FUNCTION LogMessage
VAR_INPUT
	Level : INT;
	Message : STRING;
END_VAR

IF Level >= GVLPluginFramework.LogLevel THEN
	ADSLOGSTR(	msgCtrlMask := ADSLOG_MSGTYPE_LOG, 
				msgFmtStr   := Message, 
				strArg      := '');
END_IF

END_FUNCTION

(* stored: Version 1.1.0.1, ProductVersion 3.1.4024.12
   POU LogMessage: Id {b932cb36-bcc3-4770-a9fa-39a390541f57}, SpecialFunc None *)
